{attribute 'qualified_only'}
{attribute 'strict'}
TYPE DirPlatform :
(
	
	PLUS_X := 0,
	PLUS_X_MINUS_Y := 1,
	MINUS_Y := 2,
	MINUS_X_MINUS_Y := 3,
	MINUS_X := 4,
	MINUS_X_PLUS_Y := 5,
	PLUS_Y := 6,
	PLUS_X_PLUS_Y := 7
);
END_TYPE

(* stored: Version 1.1.0.1, ProductVersion 3.1.4024.10
   DUT DirPlatform: Id {af9b4420-a1ef-4c2f-8e87-5a765d94f9f2} *)
